PROGRAM MAIN
VAR
	Axis : AXIS_REF;
	BodyExecution_AxisReset : AxesReset_Body(Axis);
	CycleExecution_AxesReset : AxesReset_Cycle(Axis);
	
END_VAR

///////////////Cycle Call for Body execution//////////////
BodyExecution_AxisReset();


///////////////Cycle Call for Cycle execution////////////
CycleExecution_AxesReset.Cycle();

END_PROGRAM

(* stored: Version 1.1.0.1, ProductVersion 3.1.4024.11
   POU MAIN: Id {43cce68e-9fd6-4b79-8662-7c36a6a087d7}, SpecialFunc None *)
